FUNCTION_BLOCK MAX_TIME (* IEC 61131-3 TIME Maximum *)
  (* Standard: 61131-3 *)
  (* Version 0.1, 2006-09-12, JHC, Holobloc Inc, Converted to Template. *)
  (* Version 0.0, 2004-12-15, JHC, Rockwell Automation, Converted from SRC format. *)
  (* Compiler header: package fb.rt.plc.select; *)
  (* Compiler classdef: (Math.max( IN1 , IN2 )) *)
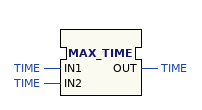
  VAR_INPUT
    IN1 : TIME;
    IN2 : TIME;
  END_VAR
  VAR_OUTPUT
    OUT : TIME; (* MAX(IN1,IN2) *)
  END_VAR
END_FUNCTION_BLOCK
